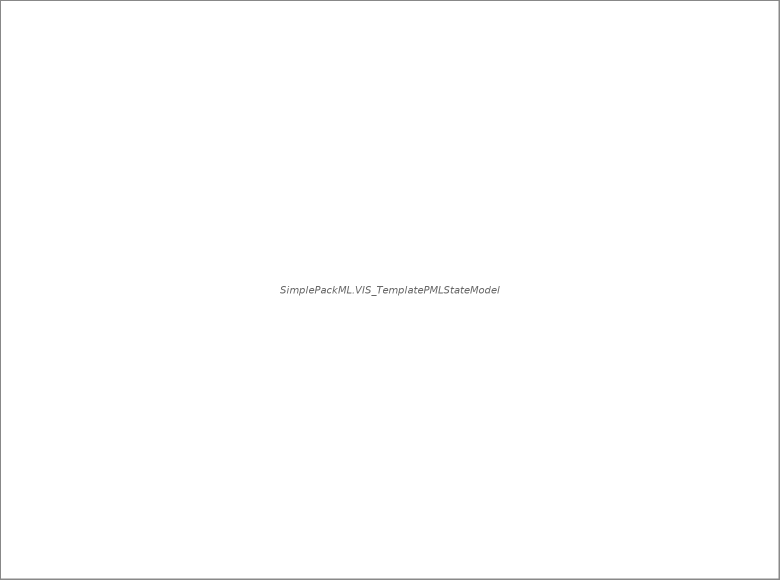
VISUALIZATION Visualization  // 780x580
    Frame (0,0 780x580)
        shows SimplePackML.VIS_TemplatePMLStateModel(ePMLUnitMode := MAIN.fbConveyor.eMode, ePMLState := MAIN.fbConveyor.eState)
END_VISUALIZATION

(* stored: Version 1.1.0.1, ProductVersion 3.1.4024.10
   Visu Visualization: Id {5f206561-9e89-4a93-b754-96610901e7bc} *)
